{attribute 'GeneratedUsingTerminal: EPP7342-0002-0016'}
{attribute addProperty BoxType "EPP7342-0002-0016"}
{attribute addProperty Id "VelocityAT %Q*INT2"}
{attribute addProperty CRC "2759475009"}
{attribute addProperty Size "2"}
TYPE DCM_Velocity_Channel_A47A3F41 :
STRUCT
	{attribute addProperty Name "Velocity"}
	Velocity AT %Q* : INT;
END_STRUCT
END_TYPE

(* stored: Version 1.2.0.0, ProductVersion 3.1.4024.9
   DUT DCM_Velocity_Channel_A47A3F41: Id {5fa2a35c-396d-4b96-a77b-6469f7a27c0c} *)
